TYPE ST_WindowTrackingTransfer :
(**************************************************************************************
 * 	Application		:	BoxControl Framework
 *	Revision		:	$Revision: 351961 $
 *	Revision date	:	$Date: 2015-07-03 16:42:43 +0200 (Fri, 03 Jul 2015) $
 *	Last changed by	:	$Author: d7mangc $
 *	URL				:	$URL: http://almscdc.swisslog.com/repo/SWPD/Development/BoxControlFramework/20_Release/trunk/01_Software/BoxControlFramework/BoxControlFramework/JumpStart/11_Library/10_Application/10_Base/F_CompareAlphaNumericString.TcPOU $
 *
 *	Purpose			:	Window tracking trasnfer data set
 *
 * ------------------------------------------------------------------------------------
 *	Copyright Swisslog [IP AG], Switzerland. All rights reserved.
 * 
 * ------------------------------------------------------------------------------------
 *	
 * 	Revision History: 
 *
 * 	VERSION			DATE			INITIALS			DESCRIPTION
 *	0.1				01.01.2001		swl					Example 
 *
 **************************************************************************************)
STRUCT
	Active					: BOOL;
	AbsoluteInsertPosition	: UDINT;
	ZoneIndex				: UINT;
	LastWindowIndex			: UINT;
END_STRUCT
END_TYPE

(* stored: Version 1.1.0.1, ProductVersion 3.1.4020.6
   DUT ST_WindowTrackingTransfer: Id {498e5aff-0e13-4873-ba44-cf50f3daf443} *)
